INTERFACE I_ProdManager

END_INTERFACE

(* stored: Version 1.1.0.1, ProductVersion 3.1.4024.11
   Itf I_ProdManager: Id {1949975c-1b60-4a62-a4e0-c6432d89843c} *)
